{attribute addProperty BoxType "EL6690-0002-0000"}
{attribute addProperty Id "StatusAT %I*Status_93A34D63810InputsEMPTY_STRUCTURE000OutputsEMPTY_STRUCTURE000WcStateAT %I*WcState_98A4DF7520.250InfoDataAT %I*InfoData_192954DE1620"}
{attribute addProperty CRC "1764312538"}
{attribute addProperty SizeInBites "26"}
{attribute addProperty SizeInBytes "3.25"}
TYPE EL6690_DEF6788A :
STRUCT
	{attribute addProperty Name "Status"}
	Status : Status_93A34D63;
	{attribute addProperty Name "Inputs"}
	Inputs : EMPTY_STRUCTURE;
	{attribute addProperty Name "Outputs"}
	Outputs : EMPTY_STRUCTURE;
	{attribute addProperty Name "WcState"}
	WcState : WcState_98A4DF75;
	{attribute addProperty Name "InfoData"}
	InfoData : InfoData_192954DE;
END_STRUCT
END_TYPE

(* stored: Version 1.2.0.0, ProductVersion 3.1.4024.9
   DUT EL6690_DEF6788A: Id {8bed97e4-ec76-4ac8-99cb-981b3c393c3b} *)
